// TIA Portal V18 export
DATA_BLOCK "数据块_2"   // DB3
{ S7_Optimized_Access := 'TRUE' }
VERSION : 0.1
// stored: AutoNumber true, DBAccessibleFromOPCUA true, IsOnlyStoredInLoadMemory false, IsRetainMemResEnabled false, IsWriteProtectedInAS false, MemoryReserve 100
   VAR
      "F-DI_A21_1" : "FIODia";   // 安全输入模块A21.1
      "F-DI_A21_2" { S7_SetPoint := 'True'} : "FIODia";   // 安全输入模块A21.2
      "F-DI_A21_3" { S7_SetPoint := 'True'} : "FIODia";   // 安全输入模块A21.3
      "F-DI_A21_4" { S7_SetPoint := 'True'} : "FIODia";   // 安全输入模块A21.4
      "F-DI_A21_5" { S7_SetPoint := 'True'} : "FIODia";   // 安全输入模块A21.5
      "F-DI_A21_6" { S7_SetPoint := 'True'} : "FIODia";   // 安全输入模块A21.6
      "F-DI_A21_7" { S7_SetPoint := 'True'} : "FIODia";   // 安全输入模块A21.7
      "F-DI_A21_8" { S7_SetPoint := 'True'} : "FIODia";   // 安全输入模块A21.8
      "F-DI_A21_9" { S7_SetPoint := 'True'} : "FIODia";   // 安全输入模块A21.9
      "F-DI_A21_10" { S7_SetPoint := 'True'} : "FIODia";   // 安全输入模块A21.10
      "F-DI_A21_11" { S7_SetPoint := 'True'} : "FIODia";   // 安全输入模块A21.11
      "F-DI_A21_12" { S7_SetPoint := 'True'} : "FIODia";   // 安全输入模块A21.12
      "F-DQ_A21_1" { S7_SetPoint := 'True'} : "FIODia";   // 安全输出模块A22.1
      "F-DQ_A21_2" { S7_SetPoint := 'True'} : "FIODia";   // 安全输出模块A22.2
   END_VAR
BEGIN
END_DATA_BLOCK
